FUNCTION_BLOCK FT_DERIV (* Calculate derivative over signal 'in' with Factor 'K' *)
  (* Standard: 61499-1 *)
  (* Version 1.0, 2025-12-19, franz *)
  PACKAGE OSCAT::Basic::POUs::Engineering::Control;
  IMPORT OSCAT::Basic::POUs::Engineering::measurements::T_PLC_US;
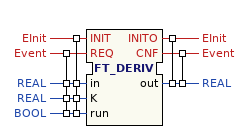
  EVENT_INPUT
    INIT : EInit WITH in, K, run; (* Init Request *)
    REQ WITH in, K, run; (* Normal Execution Request *)
  END_EVENT
  EVENT_OUTPUT
    INITO : EInit WITH out; (* Init Confirmation *)
    CNF WITH out; (* Execution Confirmation *)
  END_EVENT
  VAR_INPUT
    in : REAL; (* Input Signal *)
    K : REAL := 1.0; (* Derivation Factor *)
    run : BOOL := 1; (* Enable calculation *)
  END_VAR
  VAR_OUTPUT
    out : REAL; (* Calculated Derivative *)
  END_VAR
  VAR
    old : REAL;
    tx : DWORD;
    last : DWORD;
    init : BOOL;
    tc : REAL;
  END_VAR
  EC_STATES
    INIT : INIT -> INITO;
    REQ : REQ -> CNF;
  END_STATES
  ALGORITHM INIT IN ST:
(* Init values *)
out := 0.0;
init := FALSE;
last := 0;
old := in;
  END_ALGORITHM
  ALGORITHM REQ IN ST:
tx := T_PLC_US();
tc := DWORD_TO_REAL(tx - last);
last := tx;

(* init on first startup *)
IF NOT init THEN
	this.INIT();
	init := TRUE;
ELSIF run AND tc > 0.0 THEN
	out := (in - old) / tc * 1000000.0 * K;
	old := in;
ELSE
	out := 0.0;
END_IF;
  END_ALGORITHM
END_FUNCTION_BLOCK
